(*
Copyrights	: Precision Systems Engineering
Author		: ADBO
Date		: 07/2022
Description	: This function block is modyfication of standard FB_DoubleCoilCylinder.
It allows to operate double coil cylinder with only one sensor - active postion.
*)
FUNCTION_BLOCK FB_FixtureClamp EXTENDS FB_DoubleCoilCylinder

SUPER^();

METHOD MR_GoHome : BOOL
VAR_INPUT
END_VAR
IF eCylinderState = CYLINDER_IDLE AND piActiveSensor.In THEN
	bBusy := TRUE;
	bGoHome := TRUE;
	MR_GoHome := FALSE;
	
	eCylinderState := CYLINDER_GO_HOME;
	eCylinderGoHomeState := CYLINDER_MOVE_START_TRACKING;
	
	fbMachineLogger.MR_AddLogs(CONCAT(sName,' : home position requested'));	
	
ELSIF eCylinderState = CYLINDER_GO_HOME_DONE THEN
	bGoHome := FALSE;
	MR_GoHome := TRUE;
	
	fbMachineLogger.MR_AddLogs(CONCAT(sName,' : home position done'));	
	
END_IF
END_METHOD

METHOD PROTECTED MS_GoHome
poActiveValve.Out := FALSE;
poHomeValve.Out := TRUE;

CASE eCylinderGoHomeState OF
	CYLINDER_MOVE_START_TRACKING:
		IF NOT piActiveSensor.In THEN
			IF TIME_TO_INT(tDelay) = 0 THEN
				eCylinderGoHomeState := CYLINDER_MOVE_DONE;
			ELSE
				eCylinderGoHomeState := CYLINDER_MOVE_DELAY;
			END_IF
		END_IF
		
	CYLINDER_MOVE_DELAY:
		tonGoActiveDelay( IN := TRUE, PT := tDelay);
		
		IF tonGoActiveDelay.Q THEN
			tonGoActiveDelay( IN := FALSE );
			eCylinderGoHomeState := CYLINDER_MOVE_DONE;
		END_IF
		
	CYLINDER_MOVE_DONE:
		eCylinderState := CYLINDER_GO_HOME_DONE;
		
END_CASE
END_METHOD

END_FUNCTION_BLOCK

(* stored: Version 1.1.0.1, ProductVersion 3.1.4024.9
   POU FB_FixtureClamp: Id {2b33686c-4ffd-4fa8-be30-dab2062e7898}, SpecialFunc None
   Folder Requests: Id {0a774776-80c3-4efd-9bf7-2a6813a1e29e}
   Folder StateMachine: Id {481f6fc8-5ce0-4638-8e31-4c9ce13c27d4}
   Method MR_GoHome: Id {2a1bafef-954b-49db-90ca-a9ddf0019c85}
   Method MS_GoHome: Id {dcdf6a05-0b4d-454e-8f0f-0c0568b28ecf} *)
